{attribute 'reflection'} 
FUNCTION_BLOCK FB_Conveyor IMPLEMENTS I_SysModules
VAR
	lrVelocity 	: LREAL := 500.00;
	lrPosition 	: LREAL := 127.00;
	sStatus		: STRING := 'Running';
	
	{attribute 'instance-path'} 
    {attribute 'noinit'} 
    sPath : STRING; 
END_VAR

METHOD accept
VAR_INPUT
	iVisitor : I_Visitor;
END_VAR
iVisitor.visitConveyor(THIS^);
END_METHOD

PROPERTY pPath : STRING
GET
pPath := THIS^.sPath;
END_GET
END_PROPERTY

PROPERTY pPosition : LREAL
GET
pPosition := THIS^.lrPosition;
END_GET
END_PROPERTY

PROPERTY pStatus : STRING
GET
pStatus := THIS^.sStatus;
END_GET
END_PROPERTY

PROPERTY pVelocity : LREAL
GET
pVelocity := THIS^.lrPosition;
END_GET
END_PROPERTY

END_FUNCTION_BLOCK

(* stored: Version 1.1.0.1, ProductVersion 3.1.4024.12
   POU FB_Conveyor: Id {1f67fa7b-2adf-4297-b10d-34e2348c19bc}, SpecialFunc None
   Method accept: Id {ad644b27-f57e-48e9-8c13-9777963bd95d}
   Property pPath: Id {b88b05de-b5ac-469c-900b-57ca27b7def2}
   Get Get: Id {37b91d7f-f592-4842-b7d6-e48a33454b63}
   Property pPosition: Id {526e0903-aef9-4bd7-b0de-d71d0bcc9aad}
   Get Get: Id {1171ad54-729b-4c32-8a2d-260805486199}
   Property pStatus: Id {943cd835-d7c6-4a4a-ba91-5152ad7df583}
   Get Get: Id {8604199a-c086-47a7-95aa-5ad226d6312f}
   Property pVelocity: Id {7571d87d-5b2c-4377-a28e-1c5f9068818e}
   Get Get: Id {41ed75b4-2a96-43ea-8aad-56bc33d64688} *)
